TYPE ACRMemoryUDIntEvents :
STRUCT
	_Values : ARRAY [0..GCL.cMemoryEventsMAX] OF ACRMemoryUDIntEvent;
END_STRUCT
END_TYPE

(* stored: Version 1.1.0.1, ProductVersion 3.1.4020.12
   DUT ACRMemoryUDIntEvents: Id {f73fa50e-fd19-483d-8ce5-29fd99cc2bfc} *)
